% RSLogix 500 project project6.RSS, saved by version 8.30.00.16 %
PROJECT "UNTITLED"    % processor: Bul.1763 MicroLogix 1100 Series B %

PROGRAM FILES
  LAD 2   7 rungs

DATA FILES
  O0 OUTPUT  4 elements
  I1 INPUT  6 elements
  S2 STATUS  66 elements
  B3 BINARY  2 elements
  T4 TIMER  1 elements
  C5 COUNTER  1 elements
  R6 CONTROL  1 elements
  N7 INTEGER  4 elements
  F8 FLOAT  1 elements

LADDER 2
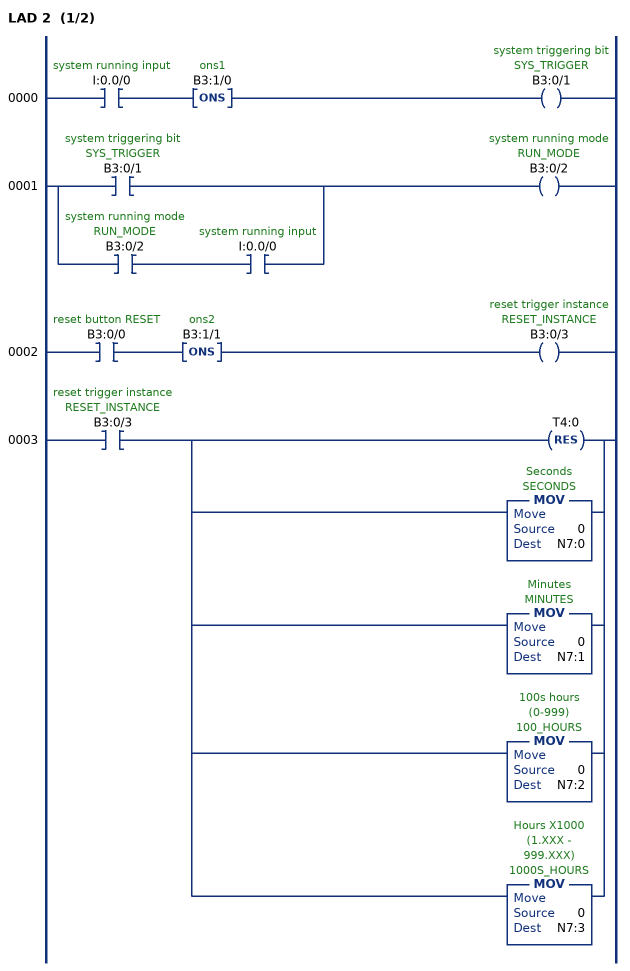
% Rung: 0 %
SOR XIC I:0.0/0 ONS B3:1/0 OTE B3:0/1 EOR
%   I:0.0/0  "system running input" %
%   B3:1/0  "ons1" %
%   B3:0/1  SYS_TRIGGER  "system triggering bit" %
% Rung: 1 %
SOR BST XIC B3:0/1 NXB XIC B3:0/2 XIC I:0.0/0 BND OTE B3:0/2 EOR
%   B3:0/1  SYS_TRIGGER  "system triggering bit" %
%   B3:0/2  RUN_MODE  "system running mode" %
%   I:0.0/0  "system running input" %
% Rung: 2 %
SOR XIC B3:0/0 ONS B3:1/1 OTE B3:0/3 EOR
%   B3:0/0  RESET  "reset button" %
%   B3:1/1  "ons2" %
%   B3:0/3  RESET_INSTANCE  "reset trigger instance" %
% Rung: 3 %
SOR XIC B3:0/3 BST RES T4:0 NXB MOV 0 N7:0 NXB MOV 0 N7:1 NXB MOV 0 N7:2 NXB MOV 0 N7:3 BND EOR
%   B3:0/3  RESET_INSTANCE  "reset trigger instance" %
%   N7:0  SECONDS  "Seconds" %
%   N7:1  MINUTES  "Minutes" %
%   N7:2  100_HOURS  "100s hours (0-999)" %
%   N7:3  1000S_HOURS  "Hours X1000 (1.XXX - 999.XXX)" %

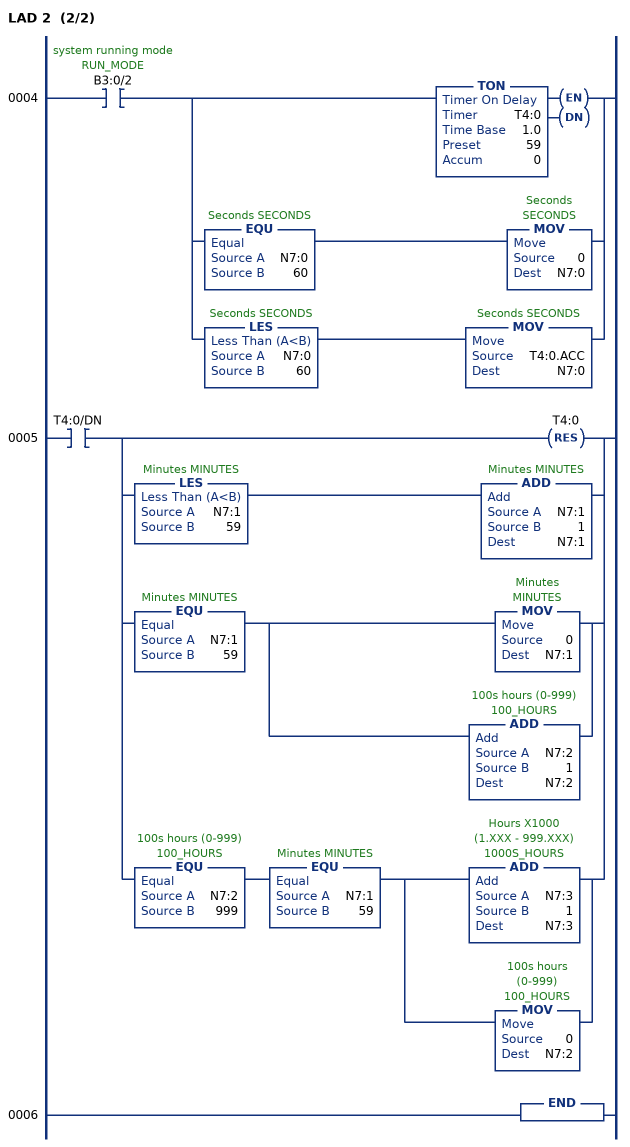
% Rung: 4 %
SOR XIC B3:0/2 BST TON T4:0 1.0 59 0 NXB EQU N7:0 60 MOV 0 N7:0 NXB LES N7:0 60 MOV T4:0.ACC N7:0 BND EOR
%   B3:0/2  RUN_MODE  "system running mode" %
%   N7:0  SECONDS  "Seconds" %
% Rung: 5 %
SOR XIC T4:0/DN BST RES T4:0 NXB LES N7:1 59 ADD N7:1 1 N7:1 NXB EQU N7:1 59 BST MOV 0 N7:1 NXB ADD N7:2 1 N7:2 BND NXB EQU N7:2 999 EQU N7:1 59 BST ADD N7:3 1 N7:3 NXB MOV 0 N7:2 BND BND EOR
%   N7:1  MINUTES  "Minutes" %
%   N7:2  100_HOURS  "100s hours (0-999)" %
%   N7:3  1000S_HOURS  "Hours X1000 (1.XXX - 999.XXX)" %
% Rung: 6 %
SOR END EOR

OTHER DOCUMENTED ADDRESSES
  C5:0  COUNTER  "seconds counter"

DATA TABLE (non-zero values as saved)
DATA T4
% .PRE .ACC %
% T4:0 % 59 0
DATA C5
% .PRE .ACC %
% C5:0 % 59 0
